FUNCTION_BLOCK FB_MotionInterlocksSync EXTENDS FB_MotionInterlocksCommon
VAR_INPUT
END_VAR
VAR_OUTPUT
END_VAR
VAR
    MotionSyncPrivateRef : REFERENCE TO FB_MotionSyncPrivate;
END_VAR

// Read external private data
IF NOT __ISVALIDREF(MotionSyncPrivateRef) THEN
    RETURN;
END_IF
// some of these vars can be used for addtional interlocks checks in
// in this class or in derived implementation
SUPER^.bReset := THIS^.MotionSyncPrivateRef.SyncPrvAbortDone;
SUPER^.bHomeBusy :=  THIS^.MotionSyncPrivateRef.SyncPrvHomeBusy;
SUPER^.bMoveBusy :=  THIS^.MotionSyncPrivateRef.SyncPrvMoveBusy;
SUPER^.bMoveDone :=  THIS^.MotionSyncPrivateRef.SyncPrvMoveDone;
SUPER^.bNewMoveReq :=  THIS^.MotionSyncPrivateRef.SyncPrvNewMoveReq;

// Call based class body
SUPER^();

// write external private data
// control MC_Power based on interlocks
THIS^.MotionSyncPrivateRef.SyncPrvAllEn := SUPER^.bAllEnabled;
THIS^.MotionSyncPrivateRef.SyncPrvAllBwdEn := SUPER^.bAllBackwardEnabled;
THIS^.MotionSyncPrivateRef.SyncPrvAllFwdEn := SUPER^.bAllForwardEnabled;
// Needed by NC homing Methods
THIS^.MotionSyncPrivateRef.SyncPrvLimBwd := SUPER^.bLimitBackwardEnable;
THIS^.MotionSyncPrivateRef.SyncPrvLimFwd := SUPER^.bLimitForwardEnable;
THIS^.MotionSyncPrivateRef.SyncPrvHome := SUPER^.bHome;

(*FB_Init is always available implicitly and it is used primarily for initialization.
The return value is not evaluated. For a specific influence, you can also declare the
methods explicitly and provide additional code there with the standard initialization
code. You can evaluate the return value.*)
METHOD FB_Init : BOOL
VAR_INPUT
    (* TRUE: the retain variables are initialized (reset warm / reset cold)*)
    bInitRetains	: BOOL;
    (* TRUE: the instance will be copied to the copy code afterward (online change)*)
    bInCopyCode	: BOOL;
    iMotionLogger	: I_MotionLogger;
    MotionSyncPrivateRef : REFERENCE TO FB_MotionSyncPrivate;
END_VAR
THIS^.MotionSyncPrivateRef REF=MotionSyncPrivateRef ;
END_METHOD

END_FUNCTION_BLOCK

(* stored: Version 1.1.0.1
   POU FB_MotionInterlocksSync: Id {31d02803-cb6f-4169-a724-4439f2f860a1}, SpecialFunc None
   Method FB_Init: Id {bbe6ed9c-a054-4a56-9a97-33c3d615425f} *)
